FUNCTION F_GetErrorsAsDWORD : DWORD
VAR_INPUT
	errStruct : DUT_Errors; 
END_VAR
VAR
	pTmp : POINTER TO DWORD;
END_VAR


pTmp := ADR(errStruct);


//pTmp := ADR(errStruct.DrahthltNichtOffen); //erstes Element von err : DUT_Errors

F_GetErrorsAsDWORD := pTmp^;

END_FUNCTION

(* stored: Version 1.1.0.1, ProductVersion 3.1.4024.3
   POU F_GetErrorsAsDWORD: Id {252b440e-f64d-44dd-8962-5b1b25ec9e28}, SpecialFunc None *)
